// TIA Portal V17 export
// export: Created 2025-03-05T07:59:20.0678202Z, ExportSetting WithDefaults, DisplayName Totally Integrated Automation Portal, DisplayVersion V17 Update 8, DisplayName TIA Portal Openness, DisplayVersion V17 Update 8, DisplayName TIA Portal Version Control Interface, DisplayVersion V17, DisplayName SINAMICS Startdrive Advanced, DisplayVersion V17 SP2, DisplayName SINAMICS Startdrive G110M, G120, G120C, G120D, G120P, G115D, DisplayVersion V17 SP2, DisplayName SINAMICS Startdrive G130, G150, S120, S150, SINAMICS MV, S210, DisplayVersion V17 SP2, DisplayName STEP 7 Professional, DisplayVersion V17 Update 8, DisplayName SINUMERIK ONE STEP 7 Toolbox, DisplayVersion V17 Update 12, DisplayName SINUMERIK 840D sl STEP 7 Toolbox, DisplayVersion V17 Update 12, DisplayName STEP 7 Safety, DisplayVersion V17 Update 6, DisplayName WinCC Advanced, DisplayVersion V17 Update 8
FUNCTION "FC7322_ROBOT_CELL_UNLOAD_FIXTURE" : Void   // FC7322, LAD
{ S7_Optimized_Access := 'FALSE' }
AUTHOR : ETXETAR
VERSION : 1.0
// stored: AutoNumber false, IsIECCheckEnabled false, SetENOAutomatically false, UDAEnableTagReadback false
   VAR_TEMP
      STATUS_BLKMOV : Int;
      TEMPORARY_Q : Any;
   END_VAR
   VAR_TEMP   // added for the SCL form of the ladder/FBD networks
      _w1 : Bool;
   END_VAR
BEGIN

REGION Network 1: >>>>>>>>>>>>>> UNIT 01 <<<<<<<<<<<<<<
END_REGION

REGION Network 2: PART A UNLOADED
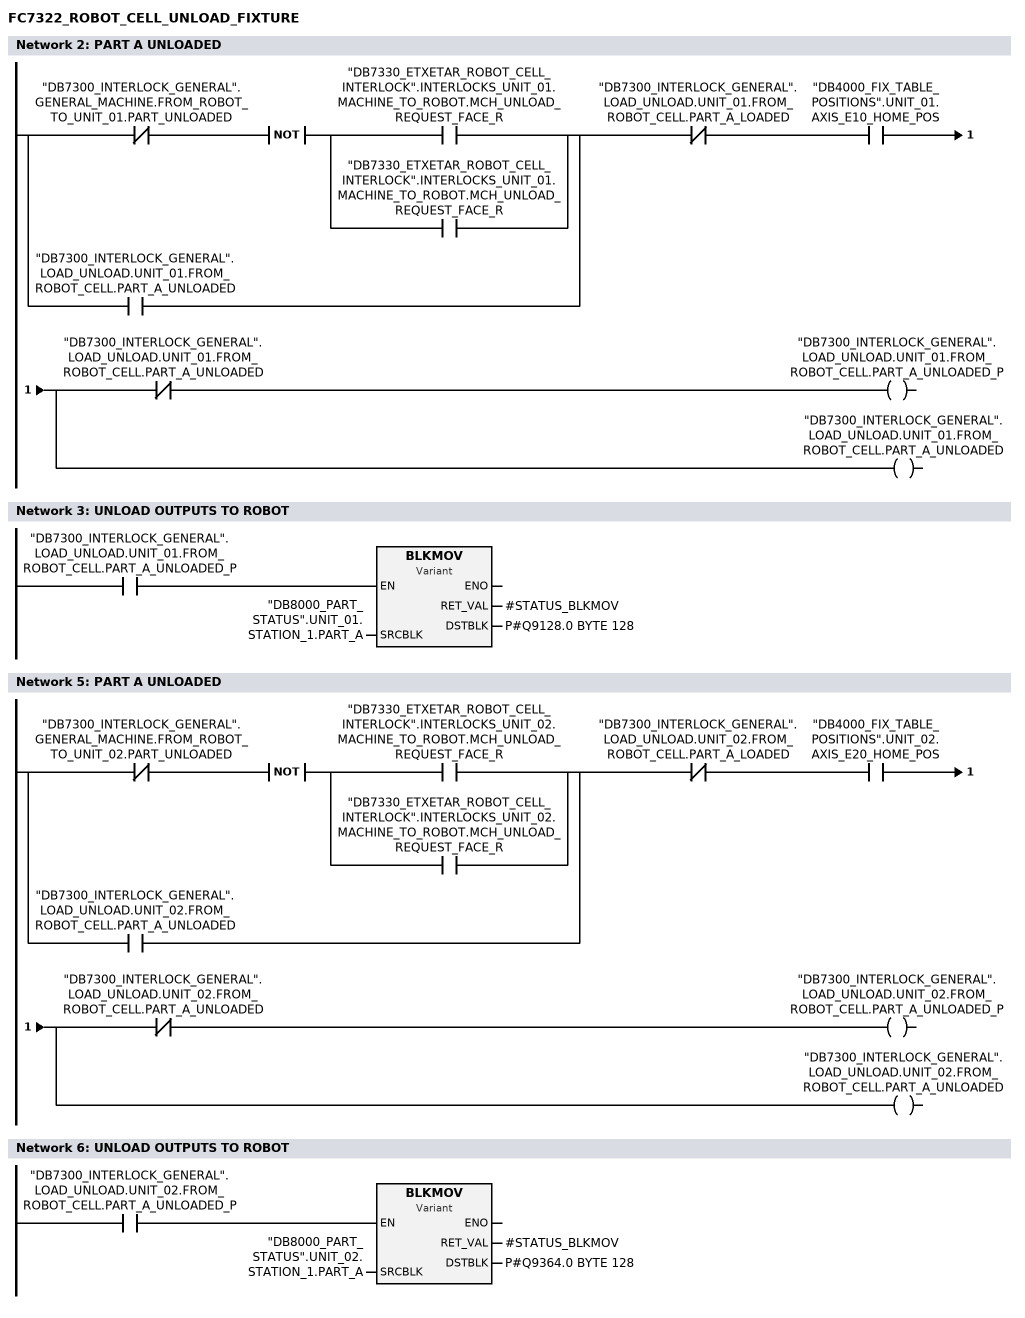
   RUNG wire#powerrail
      I_Contact( "DB7300_INTERLOCK_GENERAL".GENERAL_MACHINE.FROM_ROBOT_TO_UNIT_01.PART_UNLOADED )
      Not()
      wire#w1
      Contact( "DB7330_ETXETAR_ROBOT_CELL_INTERLOCK".INTERLOCKS_UNIT_01.MACHINE_TO_ROBOT.MCH_UNLOAD_REQUEST_FACE_R )
      wire#w2
      I_Contact( "DB7300_INTERLOCK_GENERAL".LOAD_UNLOAD.UNIT_01.FROM_ROBOT_CELL.PART_A_LOADED )
      Contact( "DB4000_FIX_TABLE_POSITIONS".UNIT_01.AXIS_E10_HOME_POS )
      wire#w3
      I_Contact( "DB7300_INTERLOCK_GENERAL".LOAD_UNLOAD.UNIT_01.FROM_ROBOT_CELL.PART_A_UNLOADED )
      Coil( "DB7300_INTERLOCK_GENERAL".LOAD_UNLOAD.UNIT_01.FROM_ROBOT_CELL.PART_A_UNLOADED_P )
   END_RUNG
   RUNG wire#w1
      Contact( "DB7330_ETXETAR_ROBOT_CELL_INTERLOCK".INTERLOCKS_UNIT_01.MACHINE_TO_ROBOT.MCH_UNLOAD_REQUEST_FACE_R )
   END_RUNG wire#w2
   RUNG wire#powerrail
      Contact( "DB7300_INTERLOCK_GENERAL".LOAD_UNLOAD.UNIT_01.FROM_ROBOT_CELL.PART_A_UNLOADED )
   END_RUNG wire#w2
   RUNG wire#w3
      Coil( "DB7300_INTERLOCK_GENERAL".LOAD_UNLOAD.UNIT_01.FROM_ROBOT_CELL.PART_A_UNLOADED )
   END_RUNG
   // the same network as SCL:
   #_w1 := ((NOT (NOT "DB7300_INTERLOCK_GENERAL".GENERAL_MACHINE.FROM_ROBOT_TO_UNIT_01.PART_UNLOADED) AND ("DB7330_ETXETAR_ROBOT_CELL_INTERLOCK".INTERLOCKS_UNIT_01.MACHINE_TO_ROBOT.MCH_UNLOAD_REQUEST_FACE_R OR "DB7330_ETXETAR_ROBOT_CELL_INTERLOCK".INTERLOCKS_UNIT_01.MACHINE_TO_ROBOT.MCH_UNLOAD_REQUEST_FACE_R)) OR "DB7300_INTERLOCK_GENERAL".LOAD_UNLOAD.UNIT_01.FROM_ROBOT_CELL.PART_A_UNLOADED) AND NOT "DB7300_INTERLOCK_GENERAL".LOAD_UNLOAD.UNIT_01.FROM_ROBOT_CELL.PART_A_LOADED AND "DB4000_FIX_TABLE_POSITIONS".UNIT_01.AXIS_E10_HOME_POS;
   "DB7300_INTERLOCK_GENERAL".LOAD_UNLOAD.UNIT_01.FROM_ROBOT_CELL.PART_A_UNLOADED_P := #_w1 AND NOT "DB7300_INTERLOCK_GENERAL".LOAD_UNLOAD.UNIT_01.FROM_ROBOT_CELL.PART_A_UNLOADED;
   "DB7300_INTERLOCK_GENERAL".LOAD_UNLOAD.UNIT_01.FROM_ROBOT_CELL.PART_A_UNLOADED := #_w1;
END_REGION

REGION Network 3: UNLOAD OUTPUTS TO ROBOT
   RUNG wire#powerrail
      Contact( "DB7300_INTERLOCK_GENERAL".LOAD_UNLOAD.UNIT_01.FROM_ROBOT_CELL.PART_A_UNLOADED_P )
      { S7_Templates := "blk_type := Variant" } BLKMOV(SRCBLK := "DB8000_PART_STATUS".UNIT_01.STATION_1.PART_A, RET_VAL => #STATUS_BLKMOV, DSTBLK => P#Q9128.0 BYTE 128)
   END_RUNG
   // the same network as SCL:
   IF "DB7300_INTERLOCK_GENERAL".LOAD_UNLOAD.UNIT_01.FROM_ROBOT_CELL.PART_A_UNLOADED_P THEN
       #STATUS_BLKMOV := BLKMOV(SRCBLK := "DB8000_PART_STATUS".UNIT_01.STATION_1.PART_A,
                               DSTBLK => P#Q9128.0 BYTE 128);
   END_IF;
END_REGION

REGION Network 4: >>>>>>>>>>>>>> UNIT 02 <<<<<<<<<<<<<<
END_REGION

REGION Network 5: PART A UNLOADED
   RUNG wire#powerrail
      I_Contact( "DB7300_INTERLOCK_GENERAL".GENERAL_MACHINE.FROM_ROBOT_TO_UNIT_02.PART_UNLOADED )
      Not()
      wire#w1
      Contact( "DB7330_ETXETAR_ROBOT_CELL_INTERLOCK".INTERLOCKS_UNIT_02.MACHINE_TO_ROBOT.MCH_UNLOAD_REQUEST_FACE_R )
      wire#w2
      I_Contact( "DB7300_INTERLOCK_GENERAL".LOAD_UNLOAD.UNIT_02.FROM_ROBOT_CELL.PART_A_LOADED )
      Contact( "DB4000_FIX_TABLE_POSITIONS".UNIT_02.AXIS_E20_HOME_POS )
      wire#w3
      I_Contact( "DB7300_INTERLOCK_GENERAL".LOAD_UNLOAD.UNIT_02.FROM_ROBOT_CELL.PART_A_UNLOADED )
      Coil( "DB7300_INTERLOCK_GENERAL".LOAD_UNLOAD.UNIT_02.FROM_ROBOT_CELL.PART_A_UNLOADED_P )
   END_RUNG
   RUNG wire#w1
      Contact( "DB7330_ETXETAR_ROBOT_CELL_INTERLOCK".INTERLOCKS_UNIT_02.MACHINE_TO_ROBOT.MCH_UNLOAD_REQUEST_FACE_R )
   END_RUNG wire#w2
   RUNG wire#powerrail
      Contact( "DB7300_INTERLOCK_GENERAL".LOAD_UNLOAD.UNIT_02.FROM_ROBOT_CELL.PART_A_UNLOADED )
   END_RUNG wire#w2
   RUNG wire#w3
      Coil( "DB7300_INTERLOCK_GENERAL".LOAD_UNLOAD.UNIT_02.FROM_ROBOT_CELL.PART_A_UNLOADED )
   END_RUNG
   // the same network as SCL:
   #_w1 := ((NOT (NOT "DB7300_INTERLOCK_GENERAL".GENERAL_MACHINE.FROM_ROBOT_TO_UNIT_02.PART_UNLOADED) AND ("DB7330_ETXETAR_ROBOT_CELL_INTERLOCK".INTERLOCKS_UNIT_02.MACHINE_TO_ROBOT.MCH_UNLOAD_REQUEST_FACE_R OR "DB7330_ETXETAR_ROBOT_CELL_INTERLOCK".INTERLOCKS_UNIT_02.MACHINE_TO_ROBOT.MCH_UNLOAD_REQUEST_FACE_R)) OR "DB7300_INTERLOCK_GENERAL".LOAD_UNLOAD.UNIT_02.FROM_ROBOT_CELL.PART_A_UNLOADED) AND NOT "DB7300_INTERLOCK_GENERAL".LOAD_UNLOAD.UNIT_02.FROM_ROBOT_CELL.PART_A_LOADED AND "DB4000_FIX_TABLE_POSITIONS".UNIT_02.AXIS_E20_HOME_POS;
   "DB7300_INTERLOCK_GENERAL".LOAD_UNLOAD.UNIT_02.FROM_ROBOT_CELL.PART_A_UNLOADED_P := #_w1 AND NOT "DB7300_INTERLOCK_GENERAL".LOAD_UNLOAD.UNIT_02.FROM_ROBOT_CELL.PART_A_UNLOADED;
   "DB7300_INTERLOCK_GENERAL".LOAD_UNLOAD.UNIT_02.FROM_ROBOT_CELL.PART_A_UNLOADED := #_w1;
END_REGION

REGION Network 6: UNLOAD OUTPUTS TO ROBOT
   RUNG wire#powerrail
      Contact( "DB7300_INTERLOCK_GENERAL".LOAD_UNLOAD.UNIT_02.FROM_ROBOT_CELL.PART_A_UNLOADED_P )
      { S7_Templates := "blk_type := Variant" } BLKMOV(SRCBLK := "DB8000_PART_STATUS".UNIT_02.STATION_1.PART_A, RET_VAL => #STATUS_BLKMOV, DSTBLK => P#Q9364.0 BYTE 128)
   END_RUNG
   // the same network as SCL:
   IF "DB7300_INTERLOCK_GENERAL".LOAD_UNLOAD.UNIT_02.FROM_ROBOT_CELL.PART_A_UNLOADED_P THEN
       #STATUS_BLKMOV := BLKMOV(SRCBLK := "DB8000_PART_STATUS".UNIT_02.STATION_1.PART_A,
                               DSTBLK => P#Q9364.0 BYTE 128);
   END_IF;
END_REGION
END_FUNCTION
